INTERFACE IComparer EXTENDS IObject

METHOD Compare : COMPARISION_RESULT
VAR_INPUT
	left : PVOID;
	right : PVOID;
END_VAR
END_METHOD

END_INTERFACE

(* stored: Version 1.1.0.1
   Itf IComparer: Id {7919720f-caf3-4677-a334-b5cdfe2e8ce5}
   Method Compare: Id {f02f14c8-397d-4c0e-8ffe-4461d30242ba} *)
